// TIA Portal V18 export
// export: Created 2026-06-08T16:04:38.4024584Z, ExportSetting WithDefaults, DisplayName Totally Integrated Automation Portal, DisplayVersion V18, DisplayName TIA Portal Openness, DisplayVersion V18, DisplayName TIA Portal Version Control Interface, DisplayVersion V18, DisplayName STEP 7 Professional, DisplayVersion V18, DisplayName STEP 7 Safety, DisplayVersion V18, DisplayName WinCC Professional, DisplayVersion V18
FUNCTION "FC_OUTPUT" : Void   // FC3, LAD
{ S7_Optimized_Access := 'TRUE' }
VERSION : 0.1
// stored: AutoNumber true, IsIECCheckEnabled false, SetENOAutomatically false, UDAEnableTagReadback false
BEGIN

REGION Network 1: BĂNG TẢI
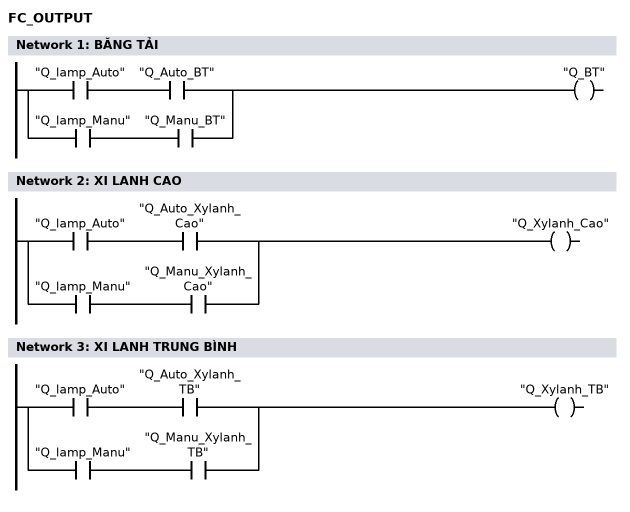
   RUNG wire#powerrail
      Contact( "Q_lamp_Auto" )
      Contact( "Q_Auto_BT" )
      wire#w1
      Coil( "Q_BT" )
   END_RUNG
   RUNG wire#powerrail
      Contact( "Q_lamp_Manu" )
      Contact( "Q_Manu_BT" )
   END_RUNG wire#w1
   // the same network as SCL:
   "Q_BT" := ("Q_lamp_Auto" AND "Q_Auto_BT") OR ("Q_lamp_Manu" AND "Q_Manu_BT");
END_REGION

REGION Network 2: XI LANH CAO
   RUNG wire#powerrail
      Contact( "Q_lamp_Auto" )
      Contact( "Q_Auto_Xylanh_Cao" )
      wire#w1
      Coil( "Q_Xylanh_Cao" )
   END_RUNG
   RUNG wire#powerrail
      Contact( "Q_lamp_Manu" )
      Contact( "Q_Manu_Xylanh_Cao" )
   END_RUNG wire#w1
   // the same network as SCL:
   "Q_Xylanh_Cao" := ("Q_lamp_Auto" AND "Q_Auto_Xylanh_Cao") OR ("Q_lamp_Manu" AND "Q_Manu_Xylanh_Cao");
END_REGION

REGION Network 3: XI LANH TRUNG BÌNH
   RUNG wire#powerrail
      Contact( "Q_lamp_Auto" )
      Contact( "Q_Auto_Xylanh_TB" )
      wire#w1
      Coil( "Q_Xylanh_TB" )
   END_RUNG
   RUNG wire#powerrail
      Contact( "Q_lamp_Manu" )
      Contact( "Q_Manu_Xylanh_TB" )
   END_RUNG wire#w1
   // the same network as SCL:
   "Q_Xylanh_TB" := ("Q_lamp_Auto" AND "Q_Auto_Xylanh_TB") OR ("Q_lamp_Manu" AND "Q_Manu_Xylanh_TB");
END_REGION
END_FUNCTION
